{attribute 'GeneratedUsingTerminal: KL3351-0003'}
{attribute addProperty BoxType "KL3351-0003"}
{attribute addProperty Id "Channel_1AT %Q*Channel_0514A8FA0"}
{attribute addProperty CRC "3350770634"}
{attribute addProperty Size "0"}
TYPE KL_C7B8B3CA :
STRUCT
	{attribute addProperty Name "Channel_1"}
	Channel_1 : Channel_0514A8FA;
END_STRUCT
END_TYPE

(* stored: Version 1.2.0.0, ProductVersion 3.1.4024.9
   DUT KL_C7B8B3CA: Id {c7c68ea5-4193-4c62-a0a0-4f2a9cac880d} *)
